// TIA Portal V20 export
DATA_BLOCK "DB_PLC_ISO_IHM"   // DB1302
{ S7_Optimized_Access := 'FALSE' }
AUTHOR : SAN
FAMILY : DPR
NAME : HMI
// stored: AutoNumber false
   VAR RETAIN
      WarmUpOn : Bool := FALSE;   // Moved to DB_HMI_Status
      KeyLaserOn : Bool := TRUE;   // Moved to DB_HMI_Status
      KeySaveParameters : Bool := FALSE;   // Not used
      bStopAfterEmptying : Bool := FALSE;   // A VOIR SI ENCORE UTILE
      Chan1_running : Bool := TRUE;   // Moved to DB_HMI_Status
      Chan2_running : Bool := FALSE;   // Moved to DB_HMI_Status
      Chan3_running : Bool := FALSE;   // Moved to DB_HMI_Status
      Chan4_running : Bool := FALSE;   // Moved to DB_HMI_Status
      StopAtNextReq { S7_SetPoint := 'True'} : Bool := FALSE;   // Moved to DB_HMI_Status
      AllChanStop : Bool := FALSE;   // Moved to DB_HMI_Status
      LoaderAutomaticMode : Bool := FALSE;   // A VOIR SI ENCORE UTILE
      LoaderManualMode : Bool := TRUE;   // A VOIR SI ENCORE UTILE
      NoCameraPresent : Bool := FALSE;   // Not used
      PremeasureZexists : Bool := FALSE;   // Not used
      PremeasureCexists : Bool := FALSE;   // Not used
      PLCFunctNotFinished : Bool := FALSE;   // Not used
      StartChangePart_station1 : Bool := FALSE;   // A VOIR SI ENCORE UTILE
      StartCheckPart_fixture1 : Bool := FALSE;   // A VOIR SI ENCORE UTILE
      Loader1PartLoad : Bool := FALSE;   // A VOIR SI ENCORE UTILE
      Loader1PartUnload : Bool := FALSE;   // A VOIR SI ENCORE UTILE
      Loader1ShiftLoad : Bool := FALSE;   // A VOIR SI ENCORE UTILE
      Loader1ShiftUnload : Bool := FALSE;   // A VOIR SI ENCORE UTILE
      Loader1LoadOpened : Bool := TRUE;   // A VOIR SI ENCORE UTILE
      Loader1UnloadOpened : Bool := TRUE;   // A VOIR SI ENCORE UTILE
      PartOnFixture1 : Bool := FALSE;   // A VOIR SI ENCORE UTILE
      MasterOnFixture1 : Bool := FALSE;   // A VOIR SI ENCORE UTILE
      StartChangePart_station2 : Bool := FALSE;   // A VOIR SI ENCORE UTILE
      StartCheckPart_fixture2 : Bool := FALSE;   // A VOIR SI ENCORE UTILE
      Loader2PartLoad : Bool := FALSE;   // A VOIR SI ENCORE UTILE
      Loader2PartUnload : Bool := FALSE;   // A VOIR SI ENCORE UTILE
      Loader2ShiftLoad : Bool := FALSE;   // A VOIR SI ENCORE UTILE
      Loader2ShiftUnload : Bool := FALSE;   // A VOIR SI ENCORE UTILE
      Loader2LoadOpened : Bool := FALSE;   // A VOIR SI ENCORE UTILE
      Loader2UnloadOpened : Bool := FALSE;   // A VOIR SI ENCORE UTILE
      PartOnFixture2 : Bool := FALSE;   // A VOIR SI ENCORE UTILE
      MasterOnFixture2 : Bool := FALSE;   // A VOIR SI ENCORE UTILE
      StartChangePart_station3 : Bool := FALSE;   // A VOIR SI ENCORE UTILE
      StartCheckPart_fixture3 : Bool := FALSE;   // A VOIR SI ENCORE UTILE
      Loader3PartLoad : Bool := FALSE;   // A VOIR SI ENCORE UTILE
      Loader3PartUnload : Bool := FALSE;   // A VOIR SI ENCORE UTILE
      Loader3ShiftLoad : Bool := FALSE;   // A VOIR SI ENCORE UTILE
      Loader3ShiftUnload : Bool := FALSE;   // A VOIR SI ENCORE UTILE
      Loader3LoadOpened : Bool := FALSE;   // A VOIR SI ENCORE UTILE
      Loader3UnloadOpened : Bool := FALSE;   // A VOIR SI ENCORE UTILE
      PartOnFixture3 : Bool := FALSE;   // A VOIR SI ENCORE UTILE
      MasterOnFixture3 : Bool := FALSE;   // A VOIR SI ENCORE UTILE
      Part_KO_go_outside_mach : Bool := TRUE;   // Not used
      MasterOnMachine : Bool := FALSE;   // Not used
      Part_position_1 : Bool := FALSE;   // A VOIR COMMENT GERER AVEC TRACABILITY
      Part_position_2 : Bool := FALSE;   // A VOIR COMMENT GERER AVEC TRACABILITY
      Part_position_3 : Bool := FALSE;   // A VOIR COMMENT GERER AVEC TRACABILITY
      Part_position_4 : Bool := FALSE;   // A VOIR COMMENT GERER AVEC TRACABILITY
      Part_position_5 : Bool := FALSE;   // A VOIR COMMENT GERER AVEC TRACABILITY
      Part_position_6 : Bool := FALSE;   // A VOIR COMMENT GERER AVEC TRACABILITY
      Part_position_7 : Bool := FALSE;   // A VOIR COMMENT GERER AVEC TRACABILITY
      Part_position_8 : Bool := FALSE;   // A VOIR COMMENT GERER AVEC TRACABILITY
      Part_position_9 : Bool := FALSE;   // A VOIR COMMENT GERER AVEC TRACABILITY
      Part_position_10 : Bool := FALSE;   // A VOIR COMMENT GERER AVEC TRACABILITY
      Part_position_11 : Bool := FALSE;   // A VOIR COMMENT GERER AVEC TRACABILITY
      Part_position_12 : Bool := FALSE;   // A VOIR COMMENT GERER AVEC TRACABILITY
      Part_position_13 : Bool := FALSE;   // A VOIR COMMENT GERER AVEC TRACABILITY
      Part_position_14 : Bool := FALSE;   // A VOIR COMMENT GERER AVEC TRACABILITY
      Part_position_15 : Bool := FALSE;   // A VOIR COMMENT GERER AVEC TRACABILITY
      Part_position_16 : Bool := FALSE;   // A VOIR COMMENT GERER AVEC TRACABILITY
      WarmUpTime : Int := 30;   // Moved to DB_HMI_Status
      Stop_For_BackWall_Wear_1 : Bool := FALSE;   // Moved to DB_HMI_Status
      Stop_For_BackWall_Wear_2 : Bool := FALSE;   // Moved to DB_HMI_Status
      Cleaning_Station_1 : Bool := FALSE;   // Moved to DB_HMI_Status
      Cleaning_Station_2 : Bool := FALSE;   // Moved to DB_HMI_Status
      Cleaning_Backwall_1 : Bool := FALSE;   // Moved to DB_HMI_Status
      Cleaning_Backwall_2 : Bool := FALSE;   // Moved to DB_HMI_Status
      Shutter_laser_closed : Bool := FALSE;   // Moved to DB_HMI_Status
      Pressure_Stop_Machine : Bool := FALSE;   // Moved to DB_HMI_Status
      Set_Bad_Part_On_Fixture : Bool := FALSE;   // Moved to DB_HMI_Status
      Reserve12 : Bool := FALSE;   // Not used
      Reserve13 : Bool := FALSE;   // Not used
      Reserve14 : Bool := FALSE;   // Not used
      Reserve15 : Bool := FALSE;   // Not used
      SemiAuto_RunEmpty : Bool := FALSE;   // A VOIR SI ENCORE UTILE
      "SemiAuto_Unload_C-Fixture" : Bool := FALSE;   // A VOIR SI ENCORE UTILE
      Reserve18 : Bool := FALSE;   // Not used
      Cnt_Washing_Loader_1 : Int := 1;   // A VOIR SI ENCORE UTILE
      Cnt_Washing_Loader_2 : Int := 0;   // A VOIR SI ENCORE UTILE
      Cnt_Part_Backwall_1 : Int := 16;   // Moved to DB_HMI_Status
      Cnt_Part_Backwall_2 : Int := 0;   // Moved to DB_HMI_Status
      Cnt_Part_Wash_Backwall_1 : Int := 26;   // Moved to DB_HMI_Status
      Cnt_Part_Wash_Backwall_2 : Int := 0;   // Moved to DB_HMI_Status
      Cnt_Part_Blow_Fixture_1 : Int;   // Moved to DB_HMI_Status
      Cnt_Part_Blow_Fixture_2 : Int;   // Moved to DB_HMI_Status
      Setpoint_laser_air_process : Real;   // Not used
      StopMachine : Bool;   // Not used
      BadPartOnFixture : Bool;   // Not used
   END_VAR
BEGIN
END_DATA_BLOCK
